FUNCTION_BLOCK FEED_CTL (* Ring Feed Control *)
  (* Standard: 61499 ITA; Classification: Testbed *)
  (* Version 0.0, 2002-05-08, JHC, Rockwell Automation *)
  (* Compiler header: package fb.rt.ita.testbed; *)
  (* Compiler Java IBM Jikes 1.06 *)
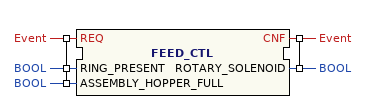
  EVENT_INPUT
    REQ WITH RING_PRESENT, ASSEMBLY_HOPPER_FULL;
  END_EVENT
  EVENT_OUTPUT
    CNF WITH ROTARY_SOLENOID;
  END_EVENT
  VAR_INPUT
    RING_PRESENT : BOOL;
    ASSEMBLY_HOPPER_FULL : BOOL;
  END_VAR
  VAR_OUTPUT
    ROTARY_SOLENOID : BOOL;
  END_VAR
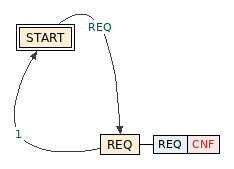
  EC_STATES
    START;
    REQ : REQ -> CNF;
  END_STATES
  EC_TRANSITIONS
    START TO REQ := REQ;
    REQ TO START := 1;
  END_TRANSITIONS
  ALGORITHM REQ IN LD:
    ROTARY_SOLENOID := RING_PRESENT  ASSEMBLY_HOPPER_FULL ! &;
  END_ALGORITHM
END_FUNCTION_BLOCK
